(* PLC project Generated.project, CODESYS CODESYS V3.5 SP19 Patch 1 *)
(* stored: creationDateTime 2026-09-06T13:00:42.496906, modificationDateTime 2026-09-06T13:00:42.496906 *)

TYPE ST_ChainTranslation : STRUCT
  Inputs_100 : ST_Chain_Translation_Inputs;
  Demandes_200 : ST_Chain_Translation_Demandes;
  Safety_300 : ST_Chain_Translation_Safety;
  Control_400 : ST_Chain_Translation_Control;
  Outputs_500 : ST_Chain_Translation_Outputs;
END_STRUCT;
END_TYPE

TYPE ST_Chain_Translation_Control : STRUCT
  Idx401_MotionAllowed : BOOL;  (* 1 = Mouvement Translation Autorisé | 0 = Bloqué *)
  Idx402_SetpointFreq_Hz : REAL;  (* [Hz] Consigne Fréquence Calculée *)
  Idx403_DriveControlWord : WORD;  (* Mot de Commande Calculé Variateur AC600 *)
  Idx404_FinalInterlockState : E_State;  (* 🛡️ État frontière *)
  Idx405_FinalInterlockReason : E_TranslationFinalInterlockReason;  (* 🛡️ Cause mémorisée *)
  Idx406_BrakeCommandOpenConfirmed : BOOL;  (* 🔌 Contacteur/bobine, pas frein mécanique *)
  Idx407_BrakeTimeoutElapsed : TIME;  (* ⏱️ Watchdog 500ms écoulé *)
END_STRUCT;
END_TYPE

TYPE ST_Chain_Translation_Demandes : STRUCT
  Idx201_JoyXRaw_ANA : INT;  (* [pts] Bruts Joystick Axe X *)
  Idx202_JoyXScaled_Pct : REAL;  (* [%] Consigne Joystick Axe X (-100% à +100%) *)
  Idx203_HmiCmd_BtnTremie : BOOL;  (* 1 = Bouton vers Trémie IHM | 0 = Relâché (ex-Idx203_HmiCmd_BtnFwd) *)
  Idx204_HmiCmd_BtnMaintenance : BOOL;  (* 1 = Bouton vers Maintenance IHM | 0 = Relâché (ex-Idx204_HmiCmd_BtnRev) *)
  Idx205_HmiTargetPosition : INT;  (* Cible Sélectionnée IHM (1=Trémie, 2=P2, 3=P1) *)
  Idx206_CycleTargetPosition : INT;  (* Cible Sélectionnée par le Cycle Auto *)
  Idx207_ModeActive : E_Mode;  (* Mode courant (MANU_N1, AUTO_N1...) *)
  Idx208_BypassNetworkActive : BOOL;  (* 0 = Comm Variateur OK | 1 = Bypass Réseau Actif ⚠️ *)
  Idx209_ArbitratedSpeed_Pct : REAL;  (* [%] Consigne finale Vitesse Translation *)
END_STRUCT;
END_TYPE

TYPE ST_Chain_Translation_Inputs : STRUCT
  Idx101_PosTremie_DI : BOOL;  (* 1 = Position Trémie Atteinte | 0 = Absent *)
  Idx102_PosPV_DI : BOOL;  (* 1 = Zone Ralentissement PV Atteinte | 0 = Absent *)
  Idx103_PosP2_DI : BOOL;  (* 1 = Position Fosse P2 Atteinte | 0 = Absent *)
  Idx104_PosP1_DI : BOOL;  (* 1 = Position Fosse P1 Atteinte | 0 = Absent *)
  Idx105_PosMaintenance_DI : BOOL;  (* 1 = Position Service Maintenance Atteinte | 0 = Absent *)
  Idx106_DriveActualFreq_Hz : REAL;  (* [Hz] Fréquence Réelle Mesurée Variateur *)
  Idx107_DriveStatusWord : WORD;  (* Mot d'état Brut Variateur AC600 *)
  Idx108_BrakeApplied : BOOL;  (* TRUE = frein SERRÉ (NOT BrakeFeedback — IHM garde le sens serré) *)
  Idx109_DriveThermalOk : BOOL;  (* TRUE = thermique moteur/variateur AC600 OK (diagnostic seul) *)
END_STRUCT;
END_TYPE

TYPE ST_Chain_Translation_Outputs : STRUCT
  Idx501_CmdDriveControlWord : WORD;  (* Mot de Commande Transmis EtherCAT AC600 *)
  Idx502_CmdDriveFreq_Hz : UINT;  (* [0.01Hz] Consigne Fréquence Transmise EtherCAT *)
  Idx503_CmdBrakeRelease_RQ : BOOL;  (* 1 = Bobine Frein Translation Alimentée (Ouvert) *)
END_STRUCT;
END_TYPE

TYPE ST_Chain_Translation_Safety : STRUCT
  Idx301_EmergencyChainClosed : BOOL;  (* 1 = Boucle Urgence OK | 0 = Arrêt d'Urgence Appuyé *)
  Idx302_SafeStopActive : BOOL;  (* 0 = Sain (Autorisé) | 1 = Arrêt Rapide Translation *)
  Idx303_PowerCutOffActive : BOOL;  (* 0 = Puissance OK | 1 = Coupure Puissance *)
  Idx304_LimitSwitchTremieActive : BOOL;  (* 0 = Sain | 1 = Fin de Course Extrême Trémie (ex-Idx304_LimitSwitchFwdActive) *)
  Idx305_LimitSwitchMaintenanceActive : BOOL;  (* 0 = Sain | 1 = Fin de Course Extrême Maintenance (ex-Idx305_LimitSwitchRevActive) *)
  Idx306_BypassLimitSwitch : BOOL;  (* 0 = Fins de course actives | 1 = Shuntés IHM ⚠️ *)
  Idx307_PositionDecoderIncoherent : BOOL;  (* 0 = Décodage 5 Capteurs OK | 1 = Incohérence Position *)
  Idx308_HeightInterlockBlocking : BOOL;  (* : 0 = M1 ET M2 ≥ hauteur mini (ou bypass) | 1 = Translation bloquée (risque collision) *)
  Idx309_ErrorOperatorComm : BOOL;  (* Défauts safety déchiffrés (bits ErrorId) — visibles individuellement à l'IHM bit0 Perte communication opérateur (joystick CAN / heartbeat IHM) *)
  Idx310_ErrorDriveComm : BOOL;  (* bit1 Perte communication EtherCAT variateur *)
  Idx311_ErrorPhaseRotation : BOOL;  (* bit2 Mauvaise rotation de phases *)
  Idx312_ErrorBrakeThermal : BOOL;  (* bit3 Surchauffe thermique frein commun *)
  Idx313_ErrorMecaB : BOOL;  (* bit4 Absence confirmation arrêt *)
  Idx314_ErrorMecaA : BOOL;  (* bit5 Mouvement non commandé *)
  Idx315_ErrorLimitSwitch : BOOL;  (* bit6 Limite extrême atteinte *)
  Idx316_ErrorSensorIncoherent : BOOL;  (* bit7 Mot capteurs position incohérent *)
  Idx317_ErrorId : WORD;  (* Masque brut complet (latch cause) — source d'arbitrage PowerCutOff *)
  Idx318_EffectivePermitM3_Tremie : BOOL;  (* Permis directionnels M3 (source unique : FB_Safety_Translation) — TRUE = autorisé, fail-safe 1 = Translation vers Trémie autorisée | 0 = SENS TRÉMIE BLOQUÉ *)
  Idx319_EffectivePermitM3_Maintenance : BOOL;  (* 1 = Translation vers Maintenance/P1 autorisée | 0 = SENS MAINTENANCE BLOQUÉ *)
END_STRUCT;
END_TYPE

(* values of E_State: DISABLED: Enable faux, neutralisé; INIT: Démarrage / vérifs; READY: Prêt, attend ordre; BUSY: Action en cours; DONE: Action terminée; STOPPING: Décél rampe avant arrêt (StartStop=FALSE ou SafeStop=TRUE); ERROR: Défaut actif non acquitté (FB en erreur — HMI non aveugle) *)

{attribute 'qualified_only'}
{attribute 'strict'}
TYPE E_State : (DISABLED := 0, INIT := 1, READY := 2, BUSY := 3, DONE := 4, STOPPING := 5, ERROR := 6);
END_TYPE

{attribute 'qualified_only'}
{attribute 'strict'}
TYPE E_TranslationFinalInterlockReason : (NONE := 0, BRAKE_COMMAND_NOT_CONFIRMED := 1, RESTART_INHIBITED := 2);
END_TYPE

(* values of E_Mode: DISABLE: Mode Désactivé / Veille de sécurité (sorties bloquées); MAINT_N1: Manuel Niveau 1 : Pilotage unitaire avec toutes sécurités actives; MAINT_N2: Manuel Niveau 2 : Pilotage dégradé (droits étendus + bypasses autorisés); SEMI_AUTO: Mode Semi-Automatique (séquenceur automatique) *)

{attribute 'qualified_only'}
{attribute 'strict'}
TYPE E_Mode : (DISABLE := 0, MAINT_N1 := 1, MAINT_N2 := 2, SEMI_AUTO := 3);
END_TYPE
